Universal Robots URScript: playera.script

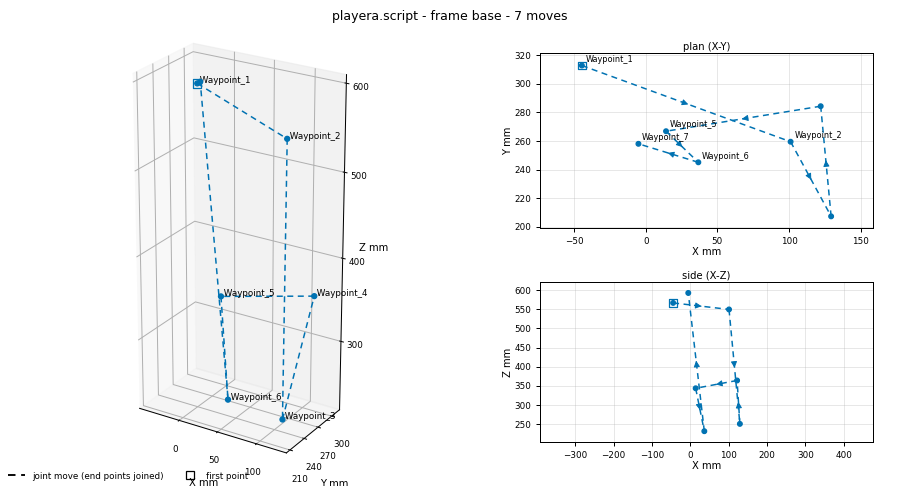
[picture p0: tool path of playera.script in frame base, 7 of 7 moves have a stored position in this frame; points joined in program order, loops and branches not executed]
def playera():
  set_tcp(p[0.0,0.0,0.0777,0.0,0.0,0.0])
  set_payload(0.1, [0.0, 0.0, 0.08])
  set_tool_voltage(24)
  set_gravity([0.0, 0.0, 9.82])
  modbus_add_signal("192.168.3.71", 255, 129, 3, "RX74", False)
  modbus_set_signal_update_frequency("RX74", 10)
  modbus_add_signal("192.168.3.133", 255, 130, 3, "TX71", False)
  modbus_set_signal_update_frequency("TX71", 10)
  modbus_set_runstate_dependent_choice("RX74",0)
  modbus_set_runstate_dependent_choice("TX71",0)
  set_standard_analog_input_domain(0, 1)
  set_standard_analog_input_domain(1, 1)
  set_tool_analog_input_domain(0, 1)
  set_tool_analog_input_domain(1, 1)
  set_analog_outputdomain(0, 0)
  set_analog_outputdomain(1, 0)
  set_input_actions_to_default()
  step_count_27ea16c7_09a7_48ac_b7d3_65c818ede42b = 0.0
  thread Step_Counter_Thread_a911c881_8547_437e_916d_f5c6adbcab51():
    while (True):
      step_count_27ea16c7_09a7_48ac_b7d3_65c818ede42b = step_count_27ea16c7_09a7_48ac_b7d3_65c818ede42b + 1.0
      sync()
    end
  end
  run Step_Counter_Thread_a911c881_8547_437e_916d_f5c6adbcab51()
  set_safety_mode_transition_hardness(1)
  global EVM=p[-0.15256820208455818,-0.42751336694884695,0.05022712170814066,-4.838863845671508E-5,-1.35928865028709E-4,-1.0092528187839596E-4]
  global EVM2=p[-0.29675101211797644,-0.4262716684008294,0.050741923201103156,4.332967508167418E-5,1.912443042895112E-4,1.5711081981983996E-4]
  global EVM3=p[0.0029371750612535727,-0.4263681938837632,0.05126173425663312,-1.739767729710799E-4,-4.4437664731219973E-5,-1.5069051907818709E-5]
  global FINAL=p[-0.22717262792356321,-0.43397417536669747,0.04266413451265917,1.4829527006895874E-4,-6.121065446531256E-5,-0.009247623504051445]
  global Plane_1=p[-0.3734029066127527,-0.3204511235418034,0.04435929145856908,9.783138506687844E-5,9.780306967539134E-5,-6.154211445520317E-5]
  global Plano4=p[-0.24996297948304783,-0.4275289861157397,0.05113872419679141,1.0348920676185259E-4,0.008007823293572955,-1.1342197607104979E-4]
  global cuervo_1=p[-0.3206063860027515,-0.4299262977046889,0.028915766646497074,-1.2221192979769074E-5,1.457304065347173E-4,-0.00918592635973644]
  global cuervo_2=p[-0.08949635923183384,-0.4299069312757706,0.028855734349918408,-2.0935967465238065E-4,-3.2568368129061994E-5,-1.9602101627311567E-4]
  global cuervo_3=p[0.1385881743231491,-0.4299379960100221,0.02888238485781129,-5.6603124500058476E-5,2.9018386427500325E-4,3.1643264082075785E-4]
  rtde_set_watchdog("speed_slider_mask", 10.0, "ignore")
  # begin: URCap Installation Node
  #   Source: OnRobot, 5.10.1, OnRobot A/S
  #   Type: Configuración de OnRobot
  # end: URCap Installation Node
  while (True):
    $ 1 "Robot Program"
    $ 2 "MoveJ"
    $ 3 "Waypoint_1" "breakAfter"
    movej(get_inverse_kin(p[-.044633714428, .312735160954, .566636518768, -1.716498950581, -.057454194109, -.032391095499], qnear=[2.616690158843994, -1.232389275227682, -1.2739341894732874, -0.9171322027789515, 0.5558661818504333, 0.1877804547548294]), a=1.3962634015954636, v=1.0471975511965976)
    $ 4 "Waypoint_2" "breakAfter"
    movej(get_inverse_kin(p[.101120173811, .259523172131, .549608262894, -1.760205805833, .318401731972, -.154282107718], qnear=[2.232118606567383, -0.9969595114337366, -1.3800528685199183, -1.1230672041522425, 0.6564516425132751, 0.3620303273200989]), a=1.3962634015954636, v=1.0471975511965976)
    $ 5 "Waypoint_3" "breakAfter"
    movej(get_inverse_kin(p[.129427566996, .207409387601, .251212344458, -2.148915414232, .206015487584, -.109101719429], qnear=[1.6846809387207031, -0.6362832228290003, -2.631979529057638, -0.48034698167909795, 1.3209930658340454, 0.17514757812023163]), a=1.3962634015954636, v=1.0471975511965976)
    $ 6 "Waypoint_4" "breakAfter"
    movej(get_inverse_kin(p[.122144694629, .284317748063, .364361076456, -1.947084601908, .195229675585, -.175783530022], qnear=[1.7568334341049194, -1.028102223073141, -2.1816399733172815, -0.3459261099444788, 1.1850241422653198, 0.1340813785791397]), a=1.3962634015954636, v=1.0471975511965976)
    $ 7 "Waypoint_5" "breakAfter"
    movej(get_inverse_kin(p[.014144168605, .266862841224, .344017942324, -1.984460664978, -.256483249116, .209794047576], qnear=[2.0953001976013184, -0.8157170454608362, -2.310735289250509, -0.44878846803774053, 1.3607653379440308, 0.1343446671962738]), a=1.3962634015954636, v=1.0471975511965976)
    $ 8 "Waypoint_6" "breakAfter"
    movej(get_inverse_kin(p[.036698124881, .245150929476, .232107249149, -2.287123753927, -.301395094147, .056343004390], qnear=[2.0612752437591553, -0.7200234572040003, -2.5861435572253626, -0.5935018698321741, 1.3488171100616455, 0.13383084535598755]), a=1.3962634015954636, v=1.0471975511965976)
    $ 9 "Waypoint_7" "breakAfter"
    movej(get_inverse_kin(p[-.005135852707, .258071249267, .592618263471, -2.021973126568, -.347522100708, .348358111854], qnear=[2.0763800144195557, -1.414469067250387, -0.5677602926837366, -1.6218183676349085, 1.5205899477005005, 0.13420122861862183]), a=1.3962634015954636, v=1.0471975511965976)
  end
end
